# B&R Automation Studio project Sh_0218_l1
Automation Studio 4.5.2.102

## Configuration Config1

CPU 4PP065.0571-P74, AutomationRuntime D4.52, Build 4.1.2, Vc V4.52.0

### Hardware
```
4PP065_0571_P74 : 4PP065.0571-P74 v1.1.2.0
  Connector IF5:
    ActivateDevice = 1
    Mode = Manual
    InternetAddress = 10.0.1.10
    SubnetMask = 255.255.255.0
  ConfigurationID = labBR
  Simulation = 1
```

## Logical view

Binary libraries used (declarations not repeated): operator, runtime, astime, AsIecCon

### Package Logical/Libraries - Global libraries

### Library Logical/Libraries/MotorCtrl (ANSIC)

#### MotorCtrl.fun - Exported functions and function blocks
```iecst
{REDUND_ERROR} FUNCTION_BLOCK FB_Integrator (*Integrator block for motor realization*) (*$GROUP=User,$CAT=User,$GROUPICON=User.png,$CATICON=User.png*)
	VAR_INPUT
		in : {REDUND_UNREPLICABLE} REAL; (*Integrator input*)
	END_VAR
	VAR_OUTPUT
		out : REAL; (*Integrator output*)
	END_VAR
	VAR
		dt : REAL; (*Step*)
	END_VAR
END_FUNCTION_BLOCK

{REDUND_ERROR} FUNCTION_BLOCK FB_Motor (*Functional block defining a motor*) (*$GROUP=User,$CAT=User,$GROUPICON=User.png,$CATICON=User.png*)
	VAR_INPUT
		u : {REDUND_UNREPLICABLE} REAL; (*Input voltage*)
	END_VAR
	VAR_OUTPUT
		w : REAL; (*Rotation frequency*)
		phi : REAL; (*Position*)
	END_VAR
	VAR
		Tm : REAL; (*Electromech constant*)
		dt : REAL; (*Step*)
		ke : REAL; (*Motor EMF *)
		first_integrator : FB_Integrator; (*Integrator*)
		second_integrator : FB_Integrator;
	END_VAR
END_FUNCTION_BLOCK

{REDUND_ERROR} FUNCTION_BLOCK FB_Regulator (*PID Regulator realization*) (*$GROUP=User,$CAT=User,$GROUPICON=User.png,$CATICON=User.png*)
	VAR_INPUT
		e : {REDUND_UNREPLICABLE} REAL; (*Difference between signal and motor rotation speed*)
	END_VAR
	VAR_OUTPUT
		u : REAL; (*Voltage going to drive input*)
	END_VAR
	VAR
		k_p : REAL; (*Proportial modifier*)
		k_i : REAL; (*Integral modifier*)
		integrator : FB_Integrator; (*Integrator*)
		iyOld : REAL; (*Previous data*)
		max_abs_value : REAL; (*Maximum edge block value*)
		dt : REAL; (*Step*)
	END_VAR
END_FUNCTION_BLOCK
```

#### FB_Integrator.c
```c
#include <bur/plctypes.h>
#ifdef __cplusplus
extern "C"
{
#endif
#include "MotorCtrl.h"
#ifdef __cplusplus
};
#endif

/* Integrator block for motor realization */

void FB_Integrator(struct FB_Integrator* inst)
{
    inst->out += inst->in*inst->dt;
}
```

#### FB_Motor.c
```c
#include <bur/plctypes.h>
#ifdef __cplusplus
extern "C"
{
#endif
#include "MotorCtrl.h"
#ifdef __cplusplus
};
#endif
/* Functional block defining a motor */
void FB_Motor(struct FB_Motor* inst)
{
    //Second integrator is used to keep 'omega' and 'phi' calcs separate
    inst->w = inst->u/inst->ke - inst->first_integrator.out;
    inst->w *= (inst->dt/inst->Tm);

    // A fucking void function and I gotta do three actions instead of one
    inst->first_integrator.in = inst->w;
    FB_Integrator(&inst->first_integrator);
    inst->w = inst->first_integrator.out;

    //Now we have 'omega' in it's final state and can compute 'phi'

    // Yeah, yeah, whatever
    inst->second_integrator.in = inst->w;
    FB_Integrator(&inst->second_integrator);
    inst->phi = inst->second_integrator.out;
}
```

#### FB_Regulator.c
```c
#include <bur/plctypes.h>
#ifdef __cplusplus
extern "C"
{
#endif
#include "MotorCtrl.h"
#ifdef __cplusplus
};
#endif
/* PID Regulator realization */

REAL voltage_limiter(REAL voltage, REAL max_voltage) {
    if (voltage > 0) {
        return (voltage > max_voltage) ? max_voltage : voltage;
    } else {
        return (voltage < -max_voltage) ? -max_voltage : voltage;
    }
}

void FB_Regulator(struct FB_Regulator* inst)
{
    REAL buffer = inst->e*inst->k_i*inst->dt + inst->iyOld;

    inst->integrator.in = buffer;
    FB_Integrator(&inst->integrator);
    buffer = inst->integrator.out;

    inst->e = voltage_limiter(inst->e * inst->k_p, inst->max_abs_value) + buffer;
    inst->u = voltage_limiter(inst->e, inst->max_abs_value);

    inst->iyOld = inst->u - inst->e;
}
```

### Program Logical/Program (ANSIC)

#### Cyclic.c - Cyclic code
```c
#include <bur/plctypes.h>

#ifdef _DEFAULT_INCLUDES
	#include <AsDefault.h>
#endif

void _CYCLIC ProgramCyclic(void)
{
	fb_regulator.e = speed;
	fb_regulator.e -= fb_motor.w;
	FB_Regulator(&fb_regulator);
	fb_motor.u = fb_regulator.u;
	FB_Motor(&fb_motor);

	secondmotor.u = speed;
	FB_Motor(&secondmotor);

	if (counter >= pwm_period){
		speed = (speed) ? 0 : 100;
		counter = 0;
	}
	counter++;
}
```

#### Init.c - Initialization code
```c
#include <bur/plctypes.h>

#ifdef _DEFAULT_INCLUDES
	#include <AsDefault.h>
#endif

void _INIT ProgramInit(void)
{
	fb_regulator.k_p = 1;
	fb_regulator.k_i = 1;
	fb_regulator.integrator.dt = 0.1;
	fb_regulator.integrator.out = 0;
	fb_regulator.iyOld = 0;
	fb_regulator.max_abs_value = 24;
	fb_regulator.dt = 0.1;

	fb_motor.phi = 0;
	fb_motor.Tm = 0.1;
	fb_motor.dt = 0.1;
	fb_motor.ke = 1;
	fb_motor.first_integrator.dt = 0.1;
	fb_motor.first_integrator.out = 0;
	fb_motor.second_integrator.dt = 0.1;
	fb_motor.second_integrator.out = 0;

	secondmotor.phi = 0;
	secondmotor.Tm = 0.1;
	secondmotor.dt = 0.1;
	secondmotor.ke = 1;
	secondmotor.first_integrator.dt = 0.1;
	secondmotor.first_integrator.out = 0;
	secondmotor.second_integrator.dt = 0.1;
	secondmotor.second_integrator.out = 0;

	speed = 100;
	pwm_period = 200;
	counter = 0;
	enable = 1;

}
```

#### Exit.c - Exit code
```c
#include <bur/plctypes.h>

#ifdef _DEFAULT_INCLUDES
#include <AsDefault.h>
#endif

void _EXIT ProgramExit(void)
{

}
```

#### Variables.var - Local variables
```iecst
VAR
	fb_regulator : FB_Regulator;
	fb_motor : FB_Motor;
	speed : REAL; (*Target speed*)
	enable : BOOL; (*ON/OFF switch*)
	pwm_period : REAL;
	counter : REAL; (*pwm switch*)
	secondmotor : FB_Motor;
END_VAR
```

Listed in the project but not available here: Logical/Global.typ, Logical/Global.var, Logical/Libraries/MotorCtrl/Types.typ, Logical/Libraries/MotorCtrl/Constants.var, Logical/Program/Types.typ
